// TIA Portal project "第一节课学习添加新设备" (V15.1)

(* hardware
DEVICE "S7-1200 station_1"  S7-1200 Station
   slot 0: "Rack_0"  S7-1200 Rack  Rack  V1.0
   slot 1: "PLC_1"  CPU 1214C DC/DC/Rly  6ES7 214-1HG40-0XB0  V4.2
   slot 2: "DI 16x24VDC_1"  SM 1221 DI16 x 24VDC  6ES7 221-1BH30-0XB0  V1.0
   slot 3: "DI 16/DQ 16x24VDC_1"  SM 1223 DI16/DQ16 x 24VDC  6ES7 223-1BL30-0XB0  V1.0
   slot 3: "DI 4x24VDC_1"  DI4 signal board (200 kHz)  6ES7 221-3BD30-0XB0  V1.0
   slot 101: "CM 1241 (RS232)_1"  6ES7 241-1AH32-0XB0  V2.2
*)

// ===== PLC "PLC_1"  CPU 1214C DC/DC/Rly =====

ORGANIZATION_BLOCK "Main"   // OB1, LAD, ProgramCycle
TITLE = "Main Program Sweep (Cycle)"
{ S7_Optimized_Access := 'TRUE' }
VERSION : 0.1
   VAR_INPUT
      Initial_Call : Bool;   // Initial call of this OB
      Remanence : Bool;   // =True, if remanent data are available
   END_VAR
BEGIN
END_ORGANIZATION_BLOCK